Staubli VAL3: showBoolStatus.pgx

public program showBoolStatus(bool x_bStatus, string& x_sEvent[])
begin
  if x_bStatus
    x_sEvent="[x]"
  else
    x_sEvent="[ ]"
  endIf
end
